FUNCTION_BLOCK Insertion2D
VAR_INPUT
	slider : I_LinearEncodedDrive;
	screw : I_LinearContinuousDrive;
END_VAR
VAR_OUTPUT
	contact AT %I* : BOOL;
	
	active : BOOL;
	error : BOOL;
	home : BOOL;
	
	homingComplete : BOOL;
	
	sliderPos : LREAL;
END_VAR
(*
this FB encapsulates 2 linear drives (1 encoded slider, 1 continuous screw) into a generic insertion machine
both drives should be declared and called externally as a concrete FB
*)

homingComplete := slider.HomeSet AND screw.HomeSet;

active := slider.Active OR screw.Active;
error := slider.Error OR screw.Error;
home := slider.AtHome AND screw.AtHome;

sliderPos := slider.CurrentPosition;

METHOD align : BOOL
VAR_INPUT
	targetPos : REAL;
END_VAR
{warning disable C0371}
slider.moveAbsolute(newTarget := targetPos);
END_METHOD

METHOD homingSequence : BOOL
VAR_INPUT
END_VAR
{warning disable C0371}
IF NOT slider.homeSet THEN
	slider.homingSequence();
END_IF

IF NOT screw.homeSet THEN
	screw.homingSequence();
END_IF

homingSequence := homingComplete;
END_METHOD

METHOD press : BOOL
VAR_INPUT
END_VAR
{warning disable C0371}
IF NOT contact THEN
	screw.moveContinuous(newDirection := MC_Negative_Direction);
END_IF
END_METHOD

METHOD release : BOOL
VAR_INPUT
END_VAR
{warning disable C0371}
screw.moveContinuous(newDirection := MC_Positive_Direction);
END_METHOD

METHOD reset : BOOL
VAR_INPUT
END_VAR
{warning disable C0371}
slider.reset();
screw.reset();
END_METHOD

METHOD stop : BOOL
VAR_INPUT
END_VAR
{warning disable C0371}
screw.stop();
slider.stop();
END_METHOD

METHOD toHome : BOOL
VAR_INPUT
END_VAR
{warning disable C0371}
slider.toHome();
screw.toHome();

toHome := slider.AtHome AND screw.AtHome;
END_METHOD

METHOD traverse : BOOL
VAR_INPUT
	direction : MC_Direction;
END_VAR
{warning disable C0371}
slider.moveContinuous(newDirection:= direction);
END_METHOD

END_FUNCTION_BLOCK

(* stored: Version 1.1.0.1, ProductVersion 3.1.4024.11
   POU Insertion2D: Id {7eea9ca1-85ea-406d-830a-7e4900221932}, SpecialFunc None
   Method align: Id {78163900-9185-402c-a1ef-d6050a8e8a9d}
   Method homingSequence: Id {1e9f95d3-ca2d-47e3-90c5-8d6354350e30}
   Method press: Id {c18f9ed0-425d-45fc-b0de-15bb8f90ec82}
   Method release: Id {83ad5159-e48f-4cd0-9425-878217c13fb1}
   Method reset: Id {7e918c71-1848-4e1f-b335-42bab28390b2}
   Method stop: Id {1b48b099-2839-4266-9926-98e0e2e28570}
   Method toHome: Id {d382636a-5273-45b3-8a46-92696ad267d2}
   Method traverse: Id {37fe2f3b-93c2-4dd6-b933-c17065052904} *)
